(* IEC 61131-3 sources: ArfBotOS/Codesys-4/ArfBotOS.fbsdev/Application.iecapp^/FUN/jog/FB_JogProcessor.fb.st^/public, 2 files *)

(* ---- M_ClearOffsets.meth.st ---- *)
METHOD PUBLIC M_ClearOffsets : BOOL
VAR_INPUT
END_VAR

FOR _j:=0 TO 3 BY 1 DO
	_OffsetExist[_j] := FALSE;
END_FOR
FOR _i := GVL_App.TCP_POS_IDX TO GVL_App.MCS_POS_IDX BY 1 DO
	StoredPositions[_i].Position.X := 0.0;
	StoredPositions[_i].Position.Y := 0.0;
	StoredPositions[_i].Position.Z := 0.0;
	StoredPositions[_i].Position.A := 0.0;
	StoredPositions[_i].Position.B := 0.0;
	StoredPositions[_i].Position.C := 0.0;
END_FOR
END_METHOD

(* ---- M_MoveToPose.meth.st ---- *)
METHOD PUBLIC M_MoveToPose : BOOL
VAR_INPUT
	Pose: E_Pose;
END_VAR

IF Enabled
	AND NOT _MoveCommandProcessor.Busy
	AND NOT _MoveCommandProcessor.Error THEN
		M_MoveToPose := TRUE;
		_MoveToPose[Pose] := TRUE;
ELSE
	M_MoveToPose := FALSE;
END_IF
END_METHOD
